FUNCTION_BLOCK PUBLIC MotorSelection
VAR_INPUT
	ManualMode: BOOL;
END_VAR
VAR
	TimeForDelay: TIME := T#0.15S;
	MovementSelection: CTUD;
	SelectionCounter: CTUD := (LOAD := TRUE, PV := 3);
	ReachedMaxSelection: BOOL;
	ReachedMinSelection: BOOL;
	UpperLeftDelay: TOF;
	UpperRightDelay: TOF;
	tmnp: TIME;
	CU: BOOL;
	CD: BOOL;
	CUU: BOOL;
	CDD: BOOL;
	PositiveEdge1: R_TRIG;
	PositiveEdge2: R_TRIG;
	temporary: BOOL;
	CUU0: BOOL;
	CDD0: BOOL;
	temporary1: BOOL;
	BURpositiveEdge: BOOL;
	BULpositiveEdge: BOOL;
	temp2: BOOL;
	temp3: BOOL;
END_VAR
VAR_OUTPUT
	CurrentSelection: INT;
END_VAR
VAR // added by the converter: edge detectors and wires of the graphical bodies
    _rt1, _rt2, _rt3, _rt4 : R_TRIG;
END_VAR

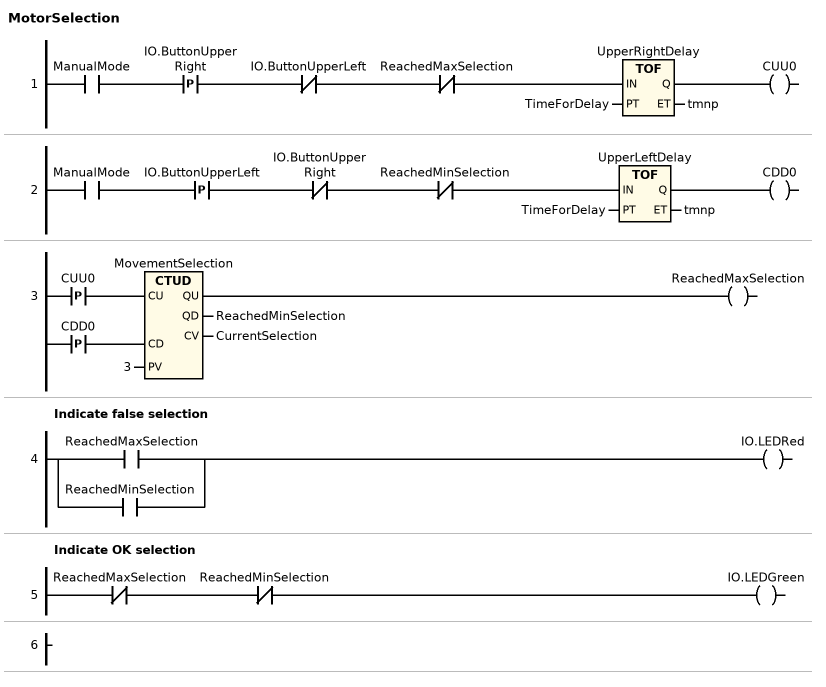
// NETWORK 1
_rt1(CLK := IO.ButtonUpperRight);
UpperRightDelay(
    IN := ManualMode AND _rt1.Q AND NOT IO.ButtonUpperLeft AND NOT ReachedMaxSelection,
    PT := TimeForDelay,
    ET => tmnp); // TOF
CUU0 := UpperRightDelay.Q;

// NETWORK 2
_rt2(CLK := IO.ButtonUpperLeft);
UpperLeftDelay(
    IN := ManualMode AND _rt2.Q AND NOT IO.ButtonUpperRight AND NOT ReachedMinSelection,
    PT := TimeForDelay,
    ET => tmnp); // TOF
CDD0 := UpperLeftDelay.Q;

// NETWORK 3
_rt3(CLK := CUU0);
_rt4(CLK := CDD0);
MovementSelection(CU := _rt3.Q, CD := _rt4.Q, PV := 3, QD => ReachedMinSelection, CV => CurrentSelection); // CTUD
ReachedMaxSelection := MovementSelection.QU;

// NETWORK 4: Indicate false selection
IO.LEDRed := ReachedMaxSelection OR ReachedMinSelection;

// NETWORK 5: Indicate OK selection
IO.LEDGreen := NOT ReachedMaxSelection AND NOT ReachedMinSelection;

// NETWORK 6

END_FUNCTION_BLOCK

(* stored: Version 1.1.0.1, ProductVersion 3.1.4024.13
   POU MotorSelection: Id {69d4fa81-a709-4d1f-a46b-7bcc0b2e8b3a}, SpecialFunc None *)
